// SIMATIC S7-200 SMART project (STEP 7-Micro/WIN SMART), CPU ST40

SYMBOL_TABLE Table 1
Timer            T101
Star             Q0.2
Delta            Q0.1
Main             Q0.0
Stop_SW          I0.1
Start_SW         I0.0
END_SYMBOL_TABLE

ORGANIZATION_BLOCK MAIN:OB1
TITLE=Program Comments
BEGIN
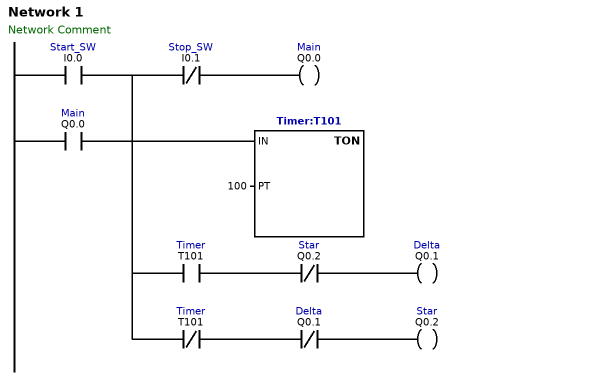
Network 1
// Network Comment
LD     Start_SW:I0.0
O      Main:Q0.0
LPS
AN     Stop_SW:I0.1
=      Main:Q0.0
LRD
TON    Timer:T101, 100
LRD
A      Timer:T101
AN     Star:Q0.2
=      Delta:Q0.1
LPP
AN     Timer:T101
AN     Delta:Q0.1
=      Star:Q0.2
END_ORGANIZATION_BLOCK
